{attribute 'qualified_only'}
{attribute 'strict'}
TYPE eTcoDriveSimpleTests :
(
    Restore := 1,
    CleanUp,
    Message,
    PowerDisable,
    PowerEnable,
    Reset,
    MoveRelativePositiveWithDisabledPositiveDirection,
    MoveRelativePositiveWithEnabledPositiveDirection,
    MoveRelativeNegativeWithDisabledNegativeDirection,
    MoveRelativeNegativeWithEnabledNegativeDirection,
    HommingDirect,
    MoveVelocityPositiveWithDisabledPositiveDirection,
    MoveVelocityPositiveWithEnabledPositiveDirection,
    Stop,
    MoveVelocityNegativeWithDisabledNegativeDirection,
    MoveVelocityNegativeWithEnabledNegativeDirection,
	MoveAbsoluteDisabled,
	MoveAbsoluteDisabledPositiveDirection,
	MoveAbsoluteEnabledPositiveDirection,
	MoveAbsoluteDisabledNegativeDirection,
	MoveAbsoluteEnabledNegativeDirection,
	
    Last
);
END_TYPE

(* stored: Version 1.1.0.1, ProductVersion 3.1.4024.12
   DUT eTcoDriveSimpleTests: Id {26cff7c3-ed2f-0d10-13fa-9a594dd7a1c9} *)
